FUNCTION_BLOCK FB81
TITLE = 'process_F2'
AUTHOR : CB

VAR
	tmp : BOOL;
END_VAR


BEGIN


NETWORK
TITLE =
//
//	process/process_F2/SyrMGT1PROC
CALL FC80 (combE := 1);
CALL FB80,	DB80;
CALL FC80 (combE := 0);




END_FUNCTION_BLOCK
